(* CoDeSys 2.3 export: ARRAYOFBYTE.EXP *)

(* Data type in STRUCT *)
TYPE ArrayOfByte :
STRUCT
	length: Length;
	items: ARRAY [0..32767] OF BYTE;
END_STRUCT
END_TYPE
